// TIA Portal V16 export
// export: Created 2022-11-24T15:20:57.6259334Z, ExportSetting WithDefaults, DisplayName Totally Integrated Automation Portal, DisplayVersion V16 Update 6, DisplayName TIA Portal Version Control Interface, DisplayVersion V16 Update 2, DisplayName TIA Portal Openness, DisplayVersion V16 Update 6, DisplayName SINAMICS Startdrive Advanced, DisplayVersion V16 Update 5, DisplayName SINAMICS Startdrive G130, G150, S120, S150, SINAMICS MV, S210, DisplayVersion V16 Update 5, DisplayName SINAMICS Startdrive G110M, G120, G120C, G120D, G120P, G115D, DisplayVersion V16 Update 5, DisplayName STEP 7 Professional, DisplayVersion V16 Update 6, DisplayName STEP 7 Safety, DisplayVersion V16, DisplayName WinCC Advanced, DisplayVersion V16 Update 6
FUNCTION "FC80_Label" : Void   // FC80, LAD
TITLE = Label device
{ S7_Optimized_Access := 'FALSE' }
VERSION : 0.1
// stored: AutoNumber false, IsIECCheckEnabled false, SetENOAutomatically false, UDAEnableTagReadback false
BEGIN

REGION Network 1: Label arm in home position for pallet transit
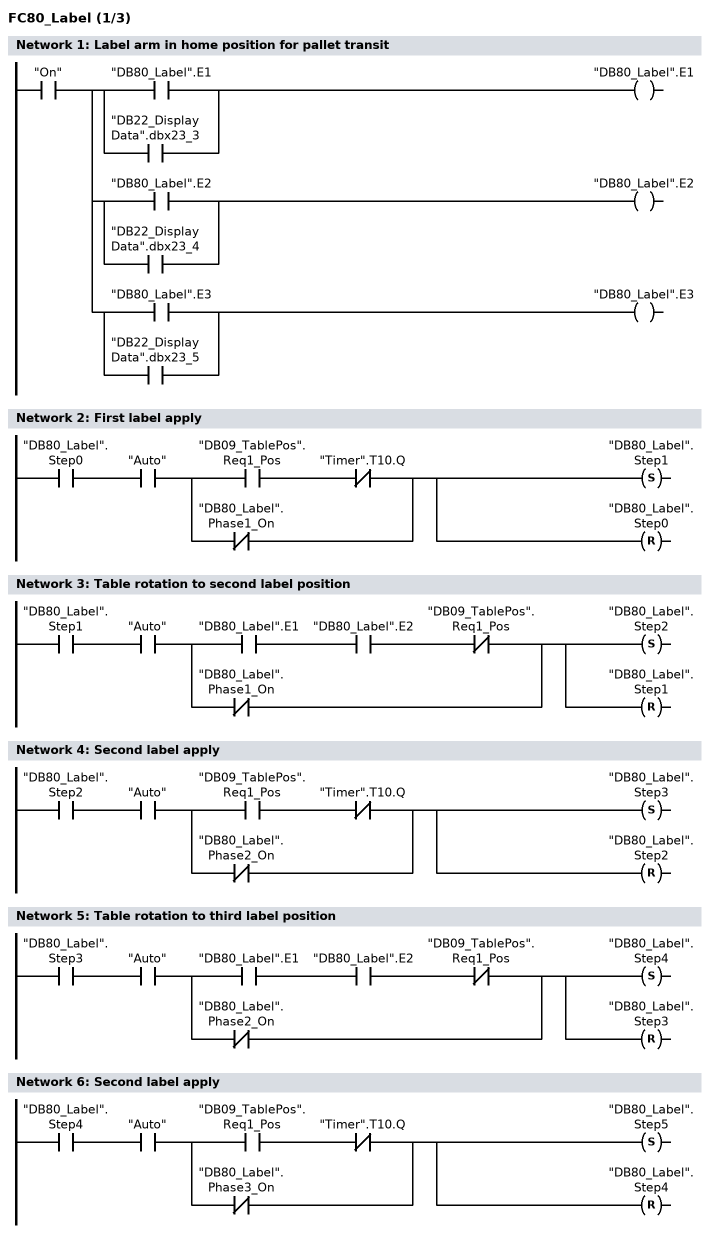
   RUNG wire#powerrail
      Contact( "On" )
      wire#w1
      Contact( "DB80_Label".E1 )
      wire#w2
      Coil( "DB80_Label".E1 )
   END_RUNG
   RUNG wire#w1
      Contact( "DB22_DisplayData".dbx23_3 )
   END_RUNG wire#w2
   RUNG wire#w1
      Contact( "DB80_Label".E2 )
      wire#w3
      Coil( "DB80_Label".E2 )
   END_RUNG
   RUNG wire#w1
      Contact( "DB22_DisplayData".dbx23_4 )
   END_RUNG wire#w3
   RUNG wire#w1
      Contact( "DB80_Label".E3 )
      wire#w4
      Coil( "DB80_Label".E3 )
   END_RUNG
   RUNG wire#w1
      Contact( "DB22_DisplayData".dbx23_5 )
   END_RUNG wire#w4
   // the same network as SCL:
   "DB80_Label".E1 := "On" AND ("DB80_Label".E1 OR "DB22_DisplayData".dbx23_3);
   "DB80_Label".E2 := "On" AND ("DB80_Label".E2 OR "DB22_DisplayData".dbx23_4);
   "DB80_Label".E3 := "On" AND ("DB80_Label".E3 OR "DB22_DisplayData".dbx23_5);
END_REGION

REGION Network 2: First label apply
   RUNG wire#powerrail
      Contact( "DB80_Label".Step0 )
      Contact( "Auto" )
      wire#w1
      Contact( "DB09_TablePos".Req1_Pos )
      I_Contact( "Timer".T10.Q )
      wire#w2
      S_Coil( "DB80_Label".Step1 )
   END_RUNG
   RUNG wire#w1
      I_Contact( "DB80_Label".Phase1_On )
   END_RUNG wire#w2
   RUNG wire#w2
      R_Coil( "DB80_Label".Step0 )
   END_RUNG
   // the same network as SCL:
   IF "DB80_Label".Step0 AND "Auto" AND (("DB09_TablePos".Req1_Pos AND NOT "Timer".T10.Q) OR NOT "DB80_Label".Phase1_On) THEN
       "DB80_Label".Step1 := TRUE;
       "DB80_Label".Step0 := FALSE;
   END_IF;
END_REGION

REGION Network 3: Table rotation to second label position
   RUNG wire#powerrail
      Contact( "DB80_Label".Step1 )
      Contact( "Auto" )
      wire#w1
      Contact( "DB80_Label".E1 )
      Contact( "DB80_Label".E2 )
      I_Contact( "DB09_TablePos".Req1_Pos )
      wire#w2
      S_Coil( "DB80_Label".Step2 )
   END_RUNG
   RUNG wire#w1
      I_Contact( "DB80_Label".Phase1_On )
   END_RUNG wire#w2
   RUNG wire#w2
      R_Coil( "DB80_Label".Step1 )
   END_RUNG
   // the same network as SCL:
   IF "DB80_Label".Step1 AND "Auto" AND (("DB80_Label".E1 AND "DB80_Label".E2 AND NOT "DB09_TablePos".Req1_Pos) OR NOT "DB80_Label".Phase1_On) THEN
       "DB80_Label".Step2 := TRUE;
       "DB80_Label".Step1 := FALSE;
   END_IF;
END_REGION

REGION Network 4: Second label apply
   RUNG wire#powerrail
      Contact( "DB80_Label".Step2 )
      Contact( "Auto" )
      wire#w1
      Contact( "DB09_TablePos".Req1_Pos )
      I_Contact( "Timer".T10.Q )
      wire#w2
      S_Coil( "DB80_Label".Step3 )
   END_RUNG
   RUNG wire#w1
      I_Contact( "DB80_Label".Phase2_On )
   END_RUNG wire#w2
   RUNG wire#w2
      R_Coil( "DB80_Label".Step2 )
   END_RUNG
   // the same network as SCL:
   IF "DB80_Label".Step2 AND "Auto" AND (("DB09_TablePos".Req1_Pos AND NOT "Timer".T10.Q) OR NOT "DB80_Label".Phase2_On) THEN
       "DB80_Label".Step3 := TRUE;
       "DB80_Label".Step2 := FALSE;
   END_IF;
END_REGION

REGION Network 5: Table rotation to third label position
   RUNG wire#powerrail
      Contact( "DB80_Label".Step3 )
      Contact( "Auto" )
      wire#w1
      Contact( "DB80_Label".E1 )
      Contact( "DB80_Label".E2 )
      I_Contact( "DB09_TablePos".Req1_Pos )
      wire#w2
      S_Coil( "DB80_Label".Step4 )
   END_RUNG
   RUNG wire#w1
      I_Contact( "DB80_Label".Phase2_On )
   END_RUNG wire#w2
   RUNG wire#w2
      R_Coil( "DB80_Label".Step3 )
   END_RUNG
   // the same network as SCL:
   IF "DB80_Label".Step3 AND "Auto" AND (("DB80_Label".E1 AND "DB80_Label".E2 AND NOT "DB09_TablePos".Req1_Pos) OR NOT "DB80_Label".Phase2_On) THEN
       "DB80_Label".Step4 := TRUE;
       "DB80_Label".Step3 := FALSE;
   END_IF;
END_REGION

REGION Network 6: Second label apply
   RUNG wire#powerrail
      Contact( "DB80_Label".Step4 )
      Contact( "Auto" )
      wire#w1
      Contact( "DB09_TablePos".Req1_Pos )
      I_Contact( "Timer".T10.Q )
      wire#w2
      S_Coil( "DB80_Label".Step5 )
   END_RUNG
   RUNG wire#w1
      I_Contact( "DB80_Label".Phase3_On )
   END_RUNG wire#w2
   RUNG wire#w2
      R_Coil( "DB80_Label".Step4 )
   END_RUNG
   // the same network as SCL:
   IF "DB80_Label".Step4 AND "Auto" AND (("DB09_TablePos".Req1_Pos AND NOT "Timer".T10.Q) OR NOT "DB80_Label".Phase3_On) THEN
       "DB80_Label".Step5 := TRUE;
       "DB80_Label".Step4 := FALSE;
   END_IF;
END_REGION

REGION Network 7: Table rotation to fourth label position
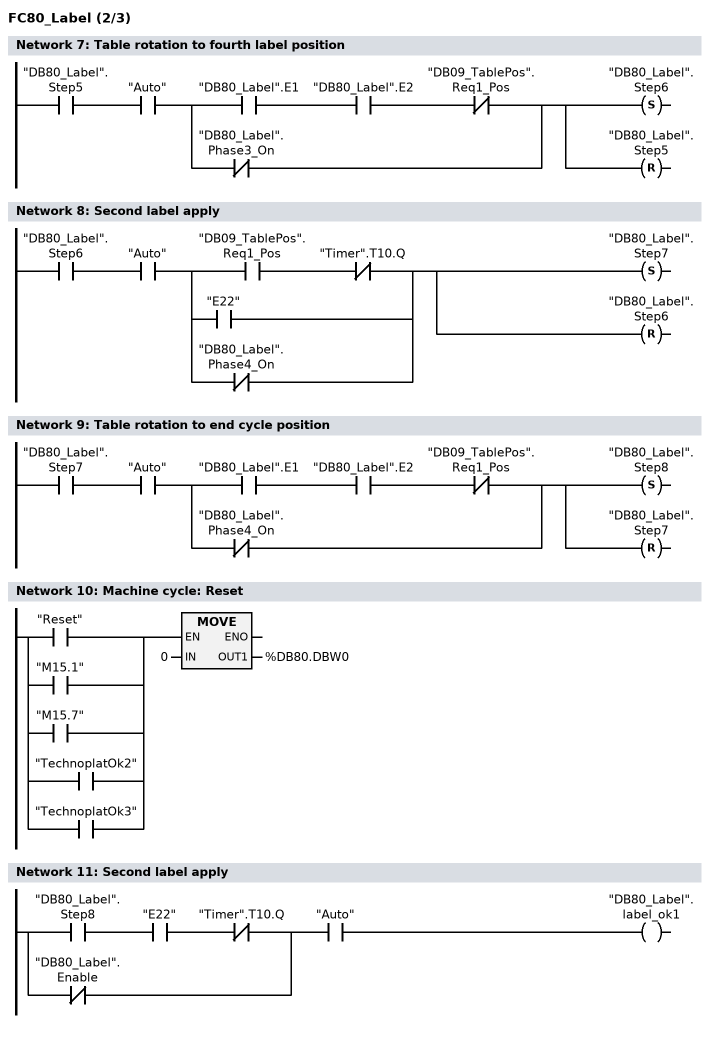
   RUNG wire#powerrail
      Contact( "DB80_Label".Step5 )
      Contact( "Auto" )
      wire#w1
      Contact( "DB80_Label".E1 )
      Contact( "DB80_Label".E2 )
      I_Contact( "DB09_TablePos".Req1_Pos )
      wire#w2
      S_Coil( "DB80_Label".Step6 )
   END_RUNG
   RUNG wire#w1
      I_Contact( "DB80_Label".Phase3_On )
   END_RUNG wire#w2
   RUNG wire#w2
      R_Coil( "DB80_Label".Step5 )
   END_RUNG
   // the same network as SCL:
   IF "DB80_Label".Step5 AND "Auto" AND (("DB80_Label".E1 AND "DB80_Label".E2 AND NOT "DB09_TablePos".Req1_Pos) OR NOT "DB80_Label".Phase3_On) THEN
       "DB80_Label".Step6 := TRUE;
       "DB80_Label".Step5 := FALSE;
   END_IF;
END_REGION

REGION Network 8: Second label apply
   RUNG wire#powerrail
      Contact( "DB80_Label".Step6 )
      Contact( "Auto" )
      wire#w1
      Contact( "DB09_TablePos".Req1_Pos )
      I_Contact( "Timer".T10.Q )
      wire#w2
      S_Coil( "DB80_Label".Step7 )
   END_RUNG
   RUNG wire#w1
      Contact( "E22" )
   END_RUNG wire#w2
   RUNG wire#w1
      I_Contact( "DB80_Label".Phase4_On )
   END_RUNG wire#w2
   RUNG wire#w2
      R_Coil( "DB80_Label".Step6 )
   END_RUNG
   // the same network as SCL:
   IF "DB80_Label".Step6 AND "Auto" AND (("DB09_TablePos".Req1_Pos AND NOT "Timer".T10.Q) OR "E22" OR NOT "DB80_Label".Phase4_On) THEN
       "DB80_Label".Step7 := TRUE;
       "DB80_Label".Step6 := FALSE;
   END_IF;
END_REGION

REGION Network 9: Table rotation to end cycle position
   RUNG wire#powerrail
      Contact( "DB80_Label".Step7 )
      Contact( "Auto" )
      wire#w1
      Contact( "DB80_Label".E1 )
      Contact( "DB80_Label".E2 )
      I_Contact( "DB09_TablePos".Req1_Pos )
      wire#w2
      S_Coil( "DB80_Label".Step8 )
   END_RUNG
   RUNG wire#w1
      I_Contact( "DB80_Label".Phase4_On )
   END_RUNG wire#w2
   RUNG wire#w2
      R_Coil( "DB80_Label".Step7 )
   END_RUNG
   // the same network as SCL:
   IF "DB80_Label".Step7 AND "Auto" AND (("DB80_Label".E1 AND "DB80_Label".E2 AND NOT "DB09_TablePos".Req1_Pos) OR NOT "DB80_Label".Phase4_On) THEN
       "DB80_Label".Step8 := TRUE;
       "DB80_Label".Step7 := FALSE;
   END_IF;
END_REGION

REGION Network 10: Machine cycle: Reset
   RUNG wire#powerrail
      Contact( "Reset" )
      wire#w1
      { S7_GenerateENO := "TRUE" } Move(in := 0, out1 => %DB80.DBW0)
   END_RUNG
   RUNG wire#powerrail
      Contact( "M15.1" )
   END_RUNG wire#w1
   RUNG wire#powerrail
      Contact( "M15.7" )
   END_RUNG wire#w1
   RUNG wire#powerrail
      Contact( "TechnoplatOk2" )
   END_RUNG wire#w1
   RUNG wire#powerrail
      Contact( "TechnoplatOk3" )
   END_RUNG wire#w1
   // the same network as SCL:
   IF "Reset" OR "M15.1" OR "M15.7" OR "TechnoplatOk2" OR "TechnoplatOk3" THEN %DB80.DBW0 := 0; END_IF;
END_REGION

REGION Network 11: Second label apply
   RUNG wire#powerrail
      Contact( "DB80_Label".Step8 )
      Contact( "E22" )
      I_Contact( "Timer".T10.Q )
      wire#w1
      Contact( "Auto" )
      Coil( "DB80_Label".label_ok1 )
   END_RUNG
   RUNG wire#powerrail
      I_Contact( "DB80_Label".Enable )
   END_RUNG wire#w1
   // the same network as SCL:
   "DB80_Label".label_ok1 := (("DB80_Label".Step8 AND "E22" AND NOT "Timer".T10.Q) OR NOT "DB80_Label".Enable) AND "Auto";
END_REGION

REGION Network 12: Label phases
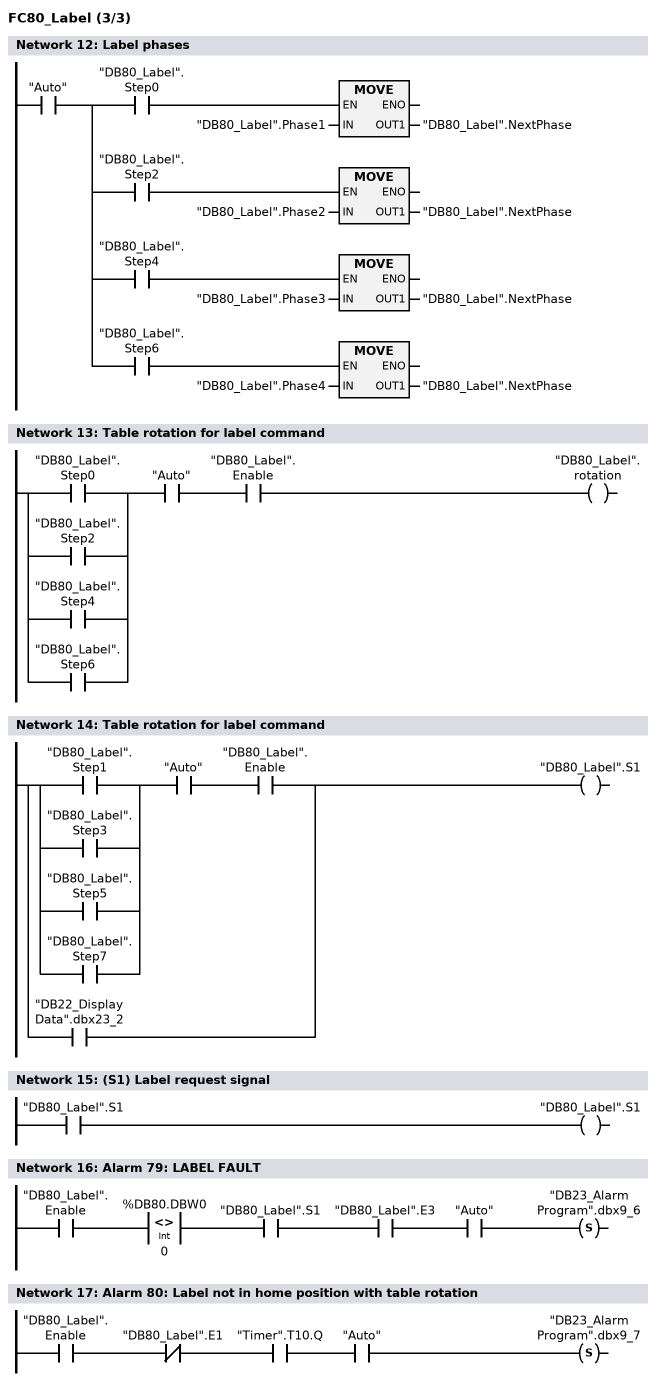
   RUNG wire#powerrail
      Contact( "Auto" )
      wire#w1
      Contact( "DB80_Label".Step0 )
      { S7_GenerateENO := "TRUE" } Move(in := "DB80_Label".Phase1, out1 => "DB80_Label".NextPhase)
   END_RUNG
   RUNG wire#w1
      Contact( "DB80_Label".Step2 )
      { S7_GenerateENO := "TRUE" } Move(in := "DB80_Label".Phase2, out1 => "DB80_Label".NextPhase)
   END_RUNG
   RUNG wire#w1
      Contact( "DB80_Label".Step4 )
      { S7_GenerateENO := "TRUE" } Move(in := "DB80_Label".Phase3, out1 => "DB80_Label".NextPhase)
   END_RUNG
   RUNG wire#w1
      Contact( "DB80_Label".Step6 )
      { S7_GenerateENO := "TRUE" } Move(in := "DB80_Label".Phase4, out1 => "DB80_Label".NextPhase)
   END_RUNG
   // the same network as SCL:
   IF "Auto" AND "DB80_Label".Step0 THEN "DB80_Label".NextPhase := "DB80_Label".Phase1; END_IF;
   IF "Auto" AND "DB80_Label".Step2 THEN "DB80_Label".NextPhase := "DB80_Label".Phase2; END_IF;
   IF "Auto" AND "DB80_Label".Step4 THEN "DB80_Label".NextPhase := "DB80_Label".Phase3; END_IF;
   IF "Auto" AND "DB80_Label".Step6 THEN "DB80_Label".NextPhase := "DB80_Label".Phase4; END_IF;
END_REGION

REGION Network 13: Table rotation for label command
   RUNG wire#powerrail
      Contact( "DB80_Label".Step0 )
      wire#w1
      Contact( "Auto" )
      Contact( "DB80_Label".Enable )
      Coil( "DB80_Label".rotation )
   END_RUNG
   RUNG wire#powerrail
      Contact( "DB80_Label".Step2 )
   END_RUNG wire#w1
   RUNG wire#powerrail
      Contact( "DB80_Label".Step4 )
   END_RUNG wire#w1
   RUNG wire#powerrail
      Contact( "DB80_Label".Step6 )
   END_RUNG wire#w1
   // the same network as SCL:
   "DB80_Label".rotation := ("DB80_Label".Step0 OR "DB80_Label".Step2 OR "DB80_Label".Step4 OR "DB80_Label".Step6) AND "Auto" AND "DB80_Label".Enable;
END_REGION

REGION Network 14: Table rotation for label command
   RUNG wire#powerrail
      Contact( "DB80_Label".Step1 )
      wire#w1
      Contact( "Auto" )
      Contact( "DB80_Label".Enable )
      wire#w2
      Coil( "DB80_Label".S1 )
   END_RUNG
   RUNG wire#powerrail
      Contact( "DB80_Label".Step3 )
   END_RUNG wire#w1
   RUNG wire#powerrail
      Contact( "DB80_Label".Step5 )
   END_RUNG wire#w1
   RUNG wire#powerrail
      Contact( "DB80_Label".Step7 )
   END_RUNG wire#w1
   RUNG wire#powerrail
      Contact( "DB22_DisplayData".dbx23_2 )
   END_RUNG wire#w2
   // the same network as SCL:
   "DB80_Label".S1 := (("DB80_Label".Step1 OR "DB80_Label".Step3 OR "DB80_Label".Step5 OR "DB80_Label".Step7) AND "Auto" AND "DB80_Label".Enable) OR "DB22_DisplayData".dbx23_2;
END_REGION

REGION Network 15: (S1) Label request signal
   RUNG wire#powerrail
      Contact( "DB80_Label".S1 )
      Coil( "DB80_Label".S1 )
   END_RUNG
   // the same network as SCL:
   "DB80_Label".S1 := "DB80_Label".S1;
END_REGION

REGION Network 16: Alarm 79: LABEL FAULT
   RUNG wire#powerrail
      Contact( "DB80_Label".Enable )
      { S7_Templates := "SrcType := Int" } NE_Contact(in1 := %DB80.DBW0, in2 := 0)
      Contact( "DB80_Label".S1 )
      Contact( "DB80_Label".E3 )
      Contact( "Auto" )
      S_Coil( "DB23_AlarmProgram".dbx9_6 )
   END_RUNG
   // the same network as SCL:
   IF "DB80_Label".Enable AND (%DB80.DBW0 <> 0) AND "DB80_Label".S1 AND "DB80_Label".E3 AND "Auto" THEN
       "DB23_AlarmProgram".dbx9_6 := TRUE;
   END_IF;
END_REGION

REGION Network 17: Alarm 80: Label not in home position with table rotation
   RUNG wire#powerrail
      Contact( "DB80_Label".Enable )
      I_Contact( "DB80_Label".E1 )
      Contact( "Timer".T10.Q )
      Contact( "Auto" )
      S_Coil( "DB23_AlarmProgram".dbx9_7 )
   END_RUNG
   // the same network as SCL:
   IF "DB80_Label".Enable AND NOT "DB80_Label".E1 AND "Timer".T10.Q AND "Auto" THEN
       "DB23_AlarmProgram".dbx9_7 := TRUE;
   END_IF;
END_REGION
END_FUNCTION
